(* Logix 5000 project; controller Text_WASH_TIMER Emulate 5570 rev 36.11; software revision 36.00 *)

TASK MainTask (continuous, watchdog 500 ms) : MainProgram, Model

MODULES
   Local : Emulate 5570 (ICP 2, rev 36.11)
       : 1756-IB16 (ICP 3, rev 3.1, Input RPI 20 ms)
       : vendor 1 type 7 code 16 (ICP 4, rev 3.1, Output RPI 20 ms)
END_MODULES

VAR_GLOBAL   (* controller tags *)
   PUSHBUTTON : ALIAS FOR Local:3:I.Data.0;   // Pushbutton Wash Cycle
   SOLENOID_CLAMP1 : ALIAS FOR Local:4:O.Data.0;   // Clamp 1 Solenoid
   SOLENOID_CLAMP2 : ALIAS FOR Local:4:O.Data.1;   // Clamp 2 Solenoid
   SWITCH_CLAMP1 : ALIAS FOR Local:3:I.Data.1;   // Limit Switch Clamp 1
   SWITCH_CLAMP2 : ALIAS FOR Local:3:I.Data.2;   // Limit Switch Clamp 2
   WASH_VALVE : ALIAS FOR Local:4:O.Data.2;   // Spray Wash Valve
END_VAR

PROGRAM MainProgram   (* main routine TextRoutine *)
VAR
   WASH_TIMER : FBD_TIMER;
END_VAR

ROUTINE TextRoutine   (* structured text *)
   //START pushbuttons to turn On/Off CLAMP solenoids
   If PUSHBUTTON then
   SOLENOID_CLAMP1[:=] 1;
   SOLENOID_CLAMP2[:=] 1;
   else;
   SOLENOID_CLAMP1:= 0;
   SOLENOID_CLAMP2:= 0;
   end_if;
   
   
   //Timer structure for time to wash
   WASH_TIMER.PRE := 5000;
   WASH_TIMER.TimerEnable :=  PUSHBUTTON & SWITCH_CLAMP1  & SWITCH_CLAMP2 ;
   TONR(WASH_TIMER);
   
   //Turn On/Off WASH valve when PUSHBUTTON and CLAMP 1 and CLAMP 2
   //switches are closed, and the time is not complete
   If PUSHBUTTON & SWITCH_CLAMP1 & SWITCH_CLAMP2 & NOT WASH_TIMER.DN  then WASH_VALVE[:=] 1;
   else;
   	WASH_VALVE:= 0;
   end_if;
END_ROUTINE
END_PROGRAM

PROGRAM Model   (* main routine Emulate *)
VAR
   HOLD : DINT;
   SOL_1_CLSD : TIMER := (PRE := 3000);
   SOL_1_OPN : TIMER := (PRE := 1000);
   SOL_2_CLSD : TIMER := (PRE := 1000);
   SOL_2_OPN : TIMER := (PRE := 2000);
END_VAR

ROUTINE Emulate   (* ladder *)
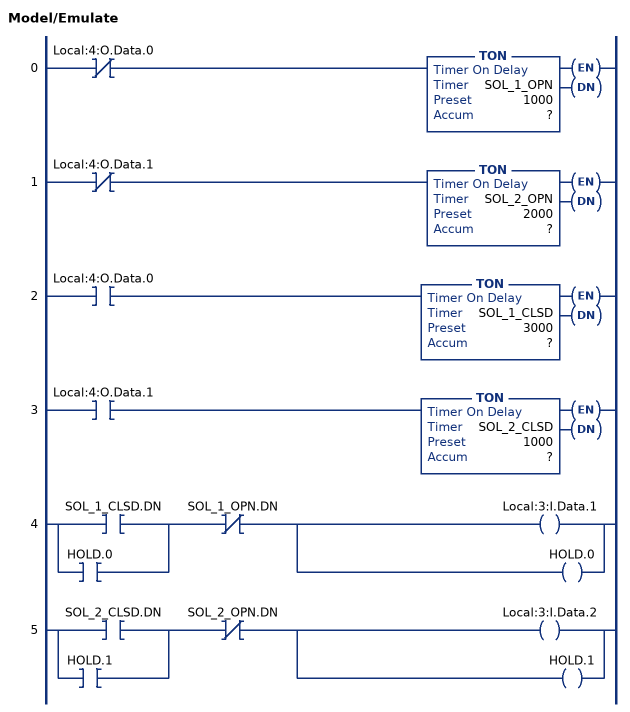
   0: XIO(Local:4:O.Data.0)TON(SOL_1_OPN,?,?);
   1: XIO(Local:4:O.Data.1)TON(SOL_2_OPN,?,?);
   2: XIC(Local:4:O.Data.0)TON(SOL_1_CLSD,?,?);
   3: XIC(Local:4:O.Data.1)TON(SOL_2_CLSD,?,?);
   4: [XIC(SOL_1_CLSD.DN) ,XIC(HOLD.0) ]XIO(SOL_1_OPN.DN)[OTE(Local:3:I.Data.1) ,OTE(HOLD.0) ];
   5: [XIC(SOL_2_CLSD.DN) ,XIC(HOLD.1) ]XIO(SOL_2_OPN.DN)[OTE(Local:3:I.Data.2) ,OTE(HOLD.1) ];
END_ROUTINE
END_PROGRAM
